// TIA Portal V19 export
DATA_BLOCK "LEDAssignment"   // DB4
{ S7_Optimized_Access := 'TRUE' }
AUTHOR : FLA
FAMILY : UHT
VERSION : 1.0
// stored: AutoNumber false, MemoryReserve 0
   VAR RETAIN
      F1_FLASH : Bool;
      F1_LIGHT : Bool;
      F2_FLASH : Bool;
      F2_LIGHT : Bool;
      F3_FLASH : Bool;
      F3_LIGHT : Bool;
      F4_FLASH : Bool;
      F4_LIGHT : Bool;
      F5_FLASH : Bool;
      F5_LIGHT : Bool;
      F6_FLASH : Bool;
      F6_LIGHT : Bool;
      F7_FLASH : Bool;
      F7_LIGHT : Bool;
      F8_FLASH : Bool;
      F8_LIGHT : Bool;
      F9_FLASH : Bool;
      F9_LIGHT : Bool;
      F10_FLASH : Bool;
      F10_LIGHT : Bool;
      F11_FLASH : Bool;
      F11_LIGHT : Bool;
      F12_FLASH : Bool;
      F12_LIGHT : Bool;
      K1_FLASH : Bool;
      K1_LIGHT : Bool;
      K2_FLASH : Bool;
      K2_LIGHT : Bool;
      K3_FLASH : Bool;
      K3_LIGHT : Bool;
      K4_FLASH : Bool;
      K4_LIGHT : Bool;
      K5_FLASH : Bool;
      K5_LIGHT : Bool;
      K6_FLASH : Bool;
      K6_LIGHT : Bool;
      K7_FLASH : Bool;
      K7_LIGHT : Bool;
      K8_FLASH : Bool;
      K8_LIGHT : Bool;
      K9_FLASH : Bool := TRUE;
      K9_LIGHT : Bool := TRUE;
      K10_FLASH : Bool;
      K10_LIGHT : Bool;
      K11_FLASH : Bool;
      K11_LIGHT : Bool;
      K12_FLASH : Bool;
      K12_LIGHT : Bool;
      K13_FLASH : Bool;
      K13_LIGHT : Bool;
      K14_FLASH : Bool;
      K14_LIGHT : Bool;
      K15_FLASH : Bool;
      K15_LIGHT : Bool;
      K16_FLASH : Bool;
      K16_LIGHT : Bool;
      SPARE_LED1 : Bool;
      SPARE_LED2 : Bool;
      SPARE_LED3 : Bool;
      SPARE_LED4 : Bool;
      SPARE_LED5 : Bool;
      SPARE_LED6 : Bool;
      SPARE_LED7 : Bool;
      SPARE_LED8 : Bool;
      SPARE_LED9 : Bool;
      SPARE_LED10 : Bool;
      SPARE_LED11 : Bool;
      SPARE_LED12 : Bool;
      SPARE_LED13 : Bool;
      SPARE_LED14 : Bool;
      SPARE_LED15 : Bool;
      SPARE_LED16 : Bool;
      SPARE_LED17 : Bool;
      SPARE_LED18 : Bool;
      SPARE_LED19 : Bool;
      SPARE_LED20 : Bool;
      SPARE_LED21 : Bool;
      SPARE_LED22 : Bool;
      SPARE_LED23 : Bool;
      SPARE_LED24 : Bool;
      F1_BUTTON : Bool;
      F2_BUTTON : Bool;
      F3_BUTTON : Bool;
      F4_BUTTON : Bool;
      F5_BUTTON : Bool;
      F6_BUTTON : Bool;
      F7_BUTTON : Bool;
      F8_BUTTON : Bool;
      F9_BUTTON : Bool;
      F10_BUTTON : Bool;
      F11_BUTTON : Bool;
      F12_BUTTON : Bool;
      F13_BUTTON : Bool;
      F14_BUTTON : Bool;
      F15_BUTTON : Bool;
      F16_BUTTON : Bool;
      F17_BUTTON : Bool;
      F18_BUTTON : Bool;
      F19_BUTTON : Bool;
      F20_BUTTON : Bool;
      K1_BUTTON : Bool;
      K2_BUTTON : Bool;
      K3_BUTTON : Bool;
      K4_BUTTON : Bool;
      K5_BUTTON : Bool;
      K6_BUTTON : Bool;
      K7_BUTTON : Bool;
      K8_BUTTON : Bool;
      K9_BUTTON : Bool;
      K10_BUTTON : Bool;
      K11_BUTTON : Bool;
      K12_BUTTON : Bool;
      K13_BUTTON : Bool;
      K14_BUTTON : Bool;
      K15_BUTTON : Bool;
      K16_BUTTON : Bool;
      SPARE_BUTTON1 : Bool;
      SPARE_BUTTON2 : Bool;
      SPARE_BUTTON3 : Bool;
      SPARE_BUTTON4 : Bool;
      SPARE_BUTTON5 : Bool;
      SPARE_BUTTON6 : Bool;
      SPARE_BUTTON7 : Bool;
      SPARE_BUTTON8 : Bool;
      SPARE_BUTTON9 : Bool;
      SPARE_BUTTON10 : Bool;
      SPARE_BUTTON11 : Bool;
      SPARE_BUTTON12 : Bool;
      ResetTotaliserHoursAHV : Bool;
      Stop_AHV_from_scada : Bool;
   END_VAR
BEGIN
END_DATA_BLOCK
